(*$
	Returns <i>TRUE</i> if the status of the instance <b><i>this</i></b> is
	<a href="#analog_actuator_status_enum"><i>ANALOG_ACTUATOR_STATUS_ACTIVE</i></a>, 
	<i>FALSE</i> otherwise.
$*)
FUNCTION analog_actuator_is_active : BOOL
VAR_IN_OUT
    CONVERSION_this:	analog_actuator;	(*$ Instance to which the method applies $*)
END_VAR

analog_actuator_is_active := (CONVERSION_this.status = ANALOG_ACTUATOR_STATUS_ACTIVE);

END_FUNCTION

(* stored: Version 1.1.0.1, ProductVersion 3.1.4022.12
   POU analog_actuator_is_active: Id {3a101f83-be59-4999-8242-1945e94a5da7}, SpecialFunc None *)
